(* IEC 61131-3 sources: Project_Icarus/backup/franzke_files, 4 files *)

(* ---- belt_out_manager.st ---- *)
PROGRAM BeltOutManager
VAR
	Step 		: DINT := 0;
	WaitTimer 	: TON;
	First		: BOOL := TRUE;
END_VAR

IF (First = TRUE)
THEN
	WaitTimer.PT := T#2S;
	WaitTimer.IN := FALSE; //Insure that there is a rising edge later
	WaitTimer();
	First := FALSE;
ELSE
	CASE (Step) OF
		0 :
			IF (PartAtBeltOut = TRUE)
			THEN
				WaitTimer.IN := FALSE;
				WaitTimer();
				BeltOutFree := FALSE;
				MotorBeltOut := TRUE;
				Step := Step + 1;
			END_IF

		1 :
			WaitTimer.IN := TRUE;
			WaitTimer();
			IF (WaitTimer.Q = TRUE)
			THEN
				WaitTimer.IN := FALSE;
				WaitTimer();
				MotorBeltOut := FALSE;
				Step := Step + 1;
			END_IF

		2 :
			IF (SensorBeltOut = TRUE)
			THEN
				MotorBeltOut := TRUE;
				Step := Step + 1;
			END_IF

		3 :
			WaitTimer.IN := TRUE;
			WaitTimer();
			IF (WaitTimer.Q = TRUE)
			THEN
				MotorBeltOut := FALSE;
				BeltOutFree := TRUE;
				Step := 0;
			END_IF

	END_CASE

END_IF

END_PROGRAM

(* ---- config.st ---- *)
VAR_CONFIG
	GVL.SliderLeft.pMotorBackward		AT	%QX32.2 : BOOL;
	GVL.SliderLeft.pMotorForward		AT	%QX32.3 : BOOL;
	GVL.SliderLeft.pSwitchBack			AT	%IX40.1 : BOOL;
	GVL.SliderLeft.pSwitchFront			AT	%IX40.0 : BOOL;

	GVL.SliderRight.pMotorBackward		AT	%QX32.4 : BOOL;
	GVL.SliderRight.pMotorForward		AT	%QX32.5 : BOOL;
	GVL.SliderRight.pSwitchBack			AT	%IX40.3 : BOOL;
	GVL.SliderRight.pSwitchFront		AT	%IX40.2 : BOOL;

	GVL.DrillingRight.pMotorBelt		AT	%QX33.1 : BOOL;
	GVL.DrillingRight.pMotorMachine		AT	%QX33.2 : BOOL;
	GVL.DrillingRight.pSensorMachine	AT	%IX40.7 : BOOL;

	GVL.DrillingLeft.pMotorBelt			AT	%QX32.7 : BOOL;
	GVL.DrillingLeft.pMotorMachine		AT	%QX33.0 : BOOL;
	GVL.DrillingLeft.pSensorMachine		AT	%IX40.5 : BOOL;

END_VAR

(* ---- drilling_manager.st ---- *)
PROGRAM DrillingManager
VAR
	First	: BOOL := TRUE;
	StepL 	: DINT := 0;
	StepR	: DINT := 0;
END_VAR

IF (First)
THEN
(*
	DrillingLeft.pMotorBelt := ADR(MotorBeltMilling);
	DrillingLeft.pMotorMachine := ADR(MotorMilling);
	DrillingLeft.pSensorMachine := ADR(SensorMilling);

	DrillingRight.pMotorBelt := ADR(MotorBeltDrilling);
	DrillingRight.pMotorMachine := ADR(MotorDrilling);
	DrillingRight.pSensorMachine := ADR(SensorDrilling);
*)
	First := FALSE;
ELSE
	DrillingLeft();
	DrillingRight();

	CASE (StepL) OF
		0 :
			DrillingLeftFree := TRUE;
			IF (PartAtDrillingL = TRUE) AND
			   (DrillingRightFree = TRUE)
			THEN
				DrillingLeftFree := FALSE;
				DrillingLeft.Start := TRUE;
				StepL := StepL + 1;
			END_IF
		1 :
			IF (DrillingLeft.Busy = TRUE) AND
			   (DrillingLeft.Done = TRUE)
			THEN
				DrillingLeft.Start := FALSE;
				PartAtDrillingR := TRUE;
				StepL := StepL + 1;
			END_IF
		2 :
			//Handshake to drilling right
			IF (DrillingRightFree = FALSE)
			THEN
				PartAtDrillingR := FALSE;
				StepL := 0;
			END_IF
	END_CASE

	CASE (StepR) OF
		0 :
			DrillingRightFree := TRUE;
			IF (PartAtDrillingR = TRUE) AND
			   (SliderRightFree = TRUE)
			THEN
				DrillingRightFree := FALSE;
				DrillingRight.Start := TRUE;
				StepR := StepR + 1;
			END_IF
		1 :
			IF (DrillingRight.Busy = TRUE) AND
			   (DrillingRight.Done = TRUE)
			THEN
				DrillingRight.Start := FALSE;
				PartAtSliderR := TRUE;
				StepR := StepR + 1;
			END_IF
		2 :
			//Handshake to slider right
			IF (SliderRightFree = FALSE)
			THEN
				PartAtSliderR := FALSE;
				StepR := 0;
			END_IF
	END_CASE

END_IF

END_PROGRAM

(* ---- slider_manager.st ---- *)
PROGRAM SliderManager
VAR
	First	: BOOL := TRUE;
	StepL	: DINT := 0;
	StepR	: DINT := 0;
END_VAR

IF (First)
THEN
(*
	SliderLeft.pMotorBackward := ADR(MotorSlider1Back);
	SliderLeft.pMotorForward := ADR(MotorSlider1Fwd);
	SliderLeft.pSwitchBack := ADR(Slider1Rear);
	SliderLeft.pSwitchFront := ADR(Slider1Front);

	SliderRight.pMotorBackward := ADR(MotorSlider2Back);
	SliderRight.pMotorForward := ADR(MotorSlider2Fwd);
	SliderRight.pSwitchBack := ADR(Slider2Rear);
	SliderRight.pSwitchFront := ADR(Slider2Front);
*)
	First := FALSE;
ELSE
	SliderLeft();
	SliderRight();

	CASE (StepL) OF
		0 :
			SliderLeftFree := TRUE;
			IF (PartAtSliderL = TRUE) AND
			   (DrillingLeftFree = TRUE) AND
			   (Slider1Rear = TRUE)
			THEN
				SliderLeftFree := FALSE;
				SliderLeft.StartForward := TRUE;
				StepL := StepL + 1;
			ELSIF (Slider1Rear = FALSE)
			THEN
				//Bring slider to base pos
				StepL := 100;
			END_IF
		1 :
			IF (SliderLeft.Busy = TRUE) AND
			   (SliderLeft.Done = TRUE)
			THEN
				SliderLeft.StartForward := FALSE;
				PartAtDrillingL := TRUE;
				StepL := StepL + 1;
			END_IF
		2 :
			SliderLeft.StartBackward := TRUE;
			StepL := StepL + 1;
		3 :
			IF (SliderLeft.Busy = TRUE) AND
			   (SliderLeft.Done = TRUE)
			THEN
				SliderLeft.StartBackward := FALSE;
				StepL := StepL + 1;
			END_IF
		4 :
			//Handshake to drilling left
			IF (DrillingLeftFree = FALSE)
			THEN
				PartAtDrillingL := FALSE;
				StepL := 0;
			END_IF
		100 :
			SliderLeft.StartBackward := TRUE;
			IF (SliderLeft.Busy = TRUE) AND
			   (SliderLeft.Done = TRUE)
			THEN
				SliderLeft.StartBackward := FALSE;
				StepL := 0;
			END_IF
	END_CASE

	CASE (StepR) OF
		0 :
			SliderRightFree := TRUE;
			IF (PartAtSliderR = TRUE) AND
			   (BeltOutFree = TRUE) AND
			   (Slider2Rear = TRUE)
			THEN
				SliderRightFree := FALSE;
				SliderRight.StartForward := TRUE;
				StepR := StepR + 1;
			ELSIF (Slider2Rear = FALSE)
			THEN
				//Bring slider to base pos
				StepR := 100;
			END_IF
		1 :
			IF (SliderRight.Busy = TRUE) AND
			   (SliderRight.Done = TRUE)
			THEN
				SliderRight.StartForward := FALSE;
				PartAtBeltOut := TRUE;
				StepR := StepR + 1;
			END_IF
		2 :
			SliderRight.StartBackward := TRUE;
			StepR := StepR + 1;
		3 :
			IF (SliderRight.Busy = TRUE) AND
			   (SliderRight.Done = TRUE)
			THEN
				SliderRight.StartBackward := FALSE;
				StepR := StepR + 1;
			END_IF
		4 :
			//Handshake to belt out
			IF (BeltOutFree = FALSE)
			THEN
				PartAtBeltOut := FALSE;
				StepR := 0;
			END_IF
		100 :
			SliderRight.StartBackward := TRUE;
			IF (SliderRight.Busy = TRUE) AND
			   (SliderRight.Done = TRUE)
			THEN
				SliderRight.StartBackward := FALSE;
				StepR := 0;
			END_IF
	END_CASE

END_IF

END_PROGRAM
